Yaskawa INFORM job: R2_ROBOTCALIB.JBI

/JOB
//NAME R2_ROBOTCALIB
///FOLDERNAME INNE
//POS
///NPOS 8,8,0,0,0,0
///TOOL 0
///POSTYPE PULSE
///PULSE
C00000=29333,-49638,-20912,73119,63857,-42959
C00001=93314,-112181,-44633,113288,19846,-54544
C00002=93177,-170797,-108894,85571,18727,-41506
C00003=29858,-67628,-75990,64239,73248,-31662
C00004=79969,53772,65947,70374,29617,-35564
C00005=114244,17686,28572,19146,13858,-9090
C00006=114151,10851,-22670,6961,41378,-3121
C00007=80801,38796,4383,38353,48218,-17598
BC00000=398161,156220,441658
BC00001=398161,156221,441652
BC00002=398161,156221,441646
BC00003=398161,156221,441643
BC00004=398161,156221,441640
BC00005=398161,156221,441638
BC00006=398161,156221,441635
BC00007=398161,156221,441632
//INST
///DATE 2023/10/04 15:13
///ATTR SC,RW
///GROUP1 RB1,BS1
NOP
MOVJ C00000 BC00000 VJ=0.78 PL=0
MOVJ C00001 BC00001 VJ=0.78 PL=0
MOVJ C00002 BC00002 VJ=0.78 PL=0
MOVJ C00003 BC00003 VJ=0.78 PL=0
MOVJ C00004 BC00004 VJ=0.78 PL=0
MOVJ C00005 BC00005 VJ=0.78 PL=0
MOVJ C00006 BC00006 VJ=0.78 PL=0
MOVJ C00007 BC00007 VJ=0.78 PL=0
END
